FUNCTION_BLOCK ARRAY2VALUES_2_LREAL (* Service Interface Function Block Type *)
  (* Description: Copyright (c) 2014 Profactor GmbH This program and the accompanying materials are made available under the terms of the Eclipse Public License 2.0 which is available at https://www.eclipse.org/legal/epl-2.0/ SPDX-License-Identifier: EPL-2.0 *)
  (* Version 1.0, 2014-07-09, Matthias Plasch, Profactor GmbH *)
  {SET_ATTRIBUTE(GenericClassName, 'GEN_ARRAY2ARRAY')}
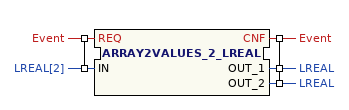
  EVENT_INPUT
    REQ WITH IN; (* Service Request *)
  END_EVENT
  EVENT_OUTPUT
    CNF WITH OUT_1, OUT_2; (* Confirmation of Requested Service *)
  END_EVENT
  VAR_INPUT
    IN : ARRAY [0..1] OF LREAL; (* Array input *)
  END_VAR
  VAR_OUTPUT
    OUT_1 : LREAL; (* output number 1 *)
    OUT_2 : LREAL; (* output number 2 *)
  END_VAR
END_FUNCTION_BLOCK
